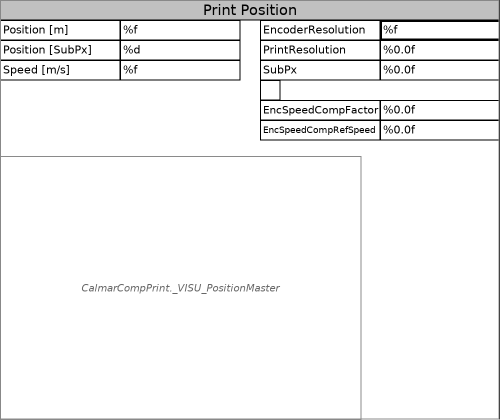
VISUALIZATION _VISU_PrintPositionDmax  // 500x420
VAR_IN_OUT
	m_Inst  : FB_PrintPositionDmax;
END_VAR
    Rectangle (0,0 500x419)
    Rectangle (0,0 500x20), "Print Position"
    Rectangle (0,20 120x20), "Position [m]"
    Rectangle (120,20 120x20), "%f", text variable: m_Inst.fbPositionMaster.fMasterPosition / 1_000_000
    Rectangle (0,40 120x20), "Position [SubPx]"
    Rectangle (120,40 120x20), "%d", text variable: m_Inst.fbPositionMaster.lMasterPosition
    Rectangle (0,60 120x20), "Speed [m/s]"
    Rectangle (120,60 120x20), "%f", text variable: m_Inst.fbPositionMaster.fMasterSpeed
    Rectangle (260,40 120x20), "PrintResolution"
    Rectangle (380,40 120x20), "%0.0f", text variable: m_Inst._fPrintResolution
    Rectangle (260,60 120x20), "SubPx"
    Rectangle (380,60 120x20), "%0.0f", text variable: m_Inst._fSubPxResolution
    Rectangle (260,20 120x20), "EncoderResolution"
    Rectangle (380,20 120x20), "%f", text variable: m_Inst._fEncoderResolution
        OnMouseClick: write the text variable via Default
    Rectangle (260,100 120x20), "EncSpeedCompFactor"
    Rectangle (380,100 120x20), "%0.0f", text variable: m_Inst._fSpeedCompFactor
    Rectangle (260,120 120x20), "EncSpeedCompRefSpeed"
    Rectangle (380,120 120x20), "%0.0f", text variable: m_Inst._fSpeedCompRefSpeed
    RoundedRectangle (260,80 20x20)
        toggle m_Inst._bEnSpeedComp
    Frame (0,156 361x264)
        shows CalmarCompPrint._VISU_PositionMaster(m_Inst_Fb := m_Inst.fbPositionMaster)
END_VISUALIZATION

(* stored: Version 1.1.0.1, ProductVersion 3.1.4024.11
   Visu _VISU_PrintPositionDmax: Id {1af8ef69-7267-4b3f-8123-ca32429a7894} *)
